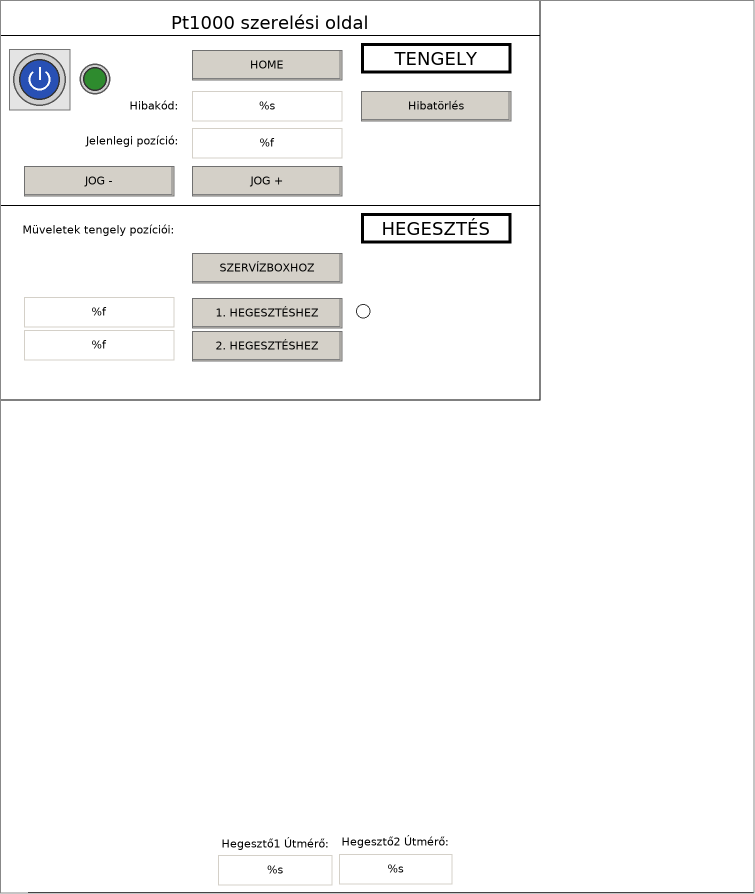
VISUALIZATION Hegesztes_Tengely_Pt1000  // 755x894
    Rectangle (0,0 540x400)
    Line (0,205) (540,205)
    Line (0,35) (540,35), "Pt1000 szerelési oldal"
    PowerSwitch (9,49 61x61), variable: GVL.bPistiServo, behaviour: TOGGLE, style: Switch-PowerSwitch-Blue
    Button (192,50 150x30), "HOME"
        OnMouseUp: execute { PISTITENGELY.sPistiAxisCommand:='HOME'; }
    Button (192,166 150x30), "JOG +"
        tap PISTITENGELY.bPistiJOGPlus
    Button (24,166 150x30), "JOG -"
        tap PISTITENGELY.bPistiJOGMinus
    Button (361,91 150x30), "Hibatörlés"
        tap PISTITENGELY.bPistiReset
    Textfield (192,91 150x30), "%s", text variable: PISTITENGELY.nPistiErrorCode, input disabled if: TRUE
    Textfield (24,330 150x30), "%f", text variable: GVL.lrHegesztoPosition7
        OnMouseClick: write the text variable via VisuDialogs.Numpad, min -10000, max -1
    Button (192,331 150x30), "2. HEGESZTÉSHEZ"
        OnMouseUp: execute { PISTITENGELY.lrPistiPosition:=GVL.lrHegesztoPosition7; PISTITENGELY.sPistiAxisCommand:='MOVE'; }
    Label (70,126 111x30), "Jelenlegi pozíció:"
    Textfield (192,128 150x30), "%f", text variable: PISTITENGELY.lrPistiActPos, input disabled if: TRUE
    RadioButton (354,253 170x116), variable: HEGESZTOK.nHegesztoNum
        Areas[0]: Text=Készenléti program
        Areas[6]: Text=6. hegesztés program
        Areas[7]: Text=7. hegesztés program
    Textfield (218,855 114x30), "%s", text variable: HEGESZTOK.ulHegeszto1Utmero, input disabled if: TRUE
    Label (200,829 150x30), "Hegesztő1 Útmérő:"
    Textfield (339,854 113x30), "%s", text variable: HEGESZTOK.ulHegeszto2Utmero, input disabled if: TRUE
    Label (320,827 150x30), "Hegesztő2 Útmérő:"
    Line (28,892) (753,892)
    Button (192,253 150x30), "SZERVÍZBOXHOZ"
        OnMouseUp: execute { PISTITENGELY.lrPistiPosition:=GVL.lrPtSzervizbox; PISTITENGELY.sPistiAxisCommand:='MOVE'; }
    Textfield (24,297 150x30), "%f", text variable: GVL.lrHegesztoPosition6
        OnMouseClick: write the text variable via VisuDialogs.Numpad, min -10000, max -1
    Button (192,298 150x30), "1. HEGESZTÉSHEZ"
        OnMouseUp: execute { PISTITENGELY.lrPistiPosition:=GVL.lrHegesztoPosition6; PISTITENGELY.sPistiAxisCommand:='MOVE'; }
    Lamp1 (77,61 36x36), variable: PISTITENGELY.bHomeReady, style: Lamp-Lamp1-Green
    Label (117,91 64x30), "Hibakód:"
    RoundedRectangle (361,43 150x30)
    Label (361,44 150x30), "TENGELY"
    RoundedRectangle (361,213 150x30)
    Label (361,214 150x30), "HEGESZTÉS"
    Label (17,215 163x30), "Müveletek tengely pozíciói:"
END_VISUALIZATION

(* stored: Version 1.1.0.1, ProductVersion 3.1.4024.11
   Visu Hegesztes_Tengely_Pt1000: Id {18cf5f8a-f465-41c2-a404-854bacf62ac9} *)
